{attribute 'linkalways'} 
{attribute 'no_explicit_call' := 'This FB is a CLASS and must be accessed using methods or properties'}
{attribute 'enable_dynamic_creation'}
FUNCTION_BLOCK Node_F_VN_VarianceFilterExp EXTENDS VisionNode
VAR
    ipSrcImage : _ITcVnImage;
    ipDestImage : _ITcVnImage;
    nKernelSize : _UDINT(0);
    fScale : _LREAL(1.0);
    eBorderType : _ETcVnBorderInterpolationMethod(ETcVnBorderInterpolationMethod.TCVN_BIM_DEFAULT);
    hrPrev : _HRESULT(S_OK);
	hresult : _HRESULT(S_OK);
END_VAR

METHOD PUBLIC  Clone : I_Node
VAR
	pNode : POINTER TO Node_F_VN_VarianceFilterExp;
END_VAR
pNode := __NEW(Node_F_VN_VarianceFilterExp);
Clone := pNode^;
END_METHOD

METHOD FB_init : BOOL
VAR_INPUT
	bInitRetains : BOOL; // if TRUE, the retain variables are initialized (warm start / cold start)
	bInCopyCode : BOOL;  // if TRUE, the instance afterwards gets moved into the copy code (online change)
END_VAR
AddInput('ipSrcImage', ipSrcImage);
AddParameter('nKernelSize', nKernelSize);
AddParameter('fScale', fScale);
AddParameter('eBorderType', eBorderType);
AddInput('hrPrev', hrPrev);
AddOutput('ipDestImage', ipDestImage);
AddOutput('hresult',hresult);
END_METHOD

METHOD PROTECTED OnExecute
hresult.Value := F_VN_VarianceFilterExp(
    ipSrcImage := ipSrcImage.Value,
	ipDestImage := ipDestImage.Value,
    nKernelSize := nKernelSize.Value,
    fScale := fScale.Value,
    eBorderType := eBorderType.Value,
	hrPrev:= hrPrev.Value);
END_METHOD

METHOD PUBLIC PreExecutionCheck
VAR_INPUT
	Check : I_PreExecutionChecks;
END_VAR
Check.IsTrue(ipSrcImage.IsValid, 'ipSrcImage must contain an image');
Check.IsTrue(ipSrcImage.HasChannelCount(1), 'ipSrcImage must have 1 channel');
Check.IsTrue(ipSrcImage.IsPixelDepth(8), 'ipSrcImage must have 8 bit pixel depth');
END_METHOD

END_FUNCTION_BLOCK

(* stored: Version 1.1.0.1, ProductVersion 3.1.4024.15
   POU Node_F_VN_VarianceFilterExp: Id {ec72eb1b-c208-0201-29da-b8ee69a8bbda}, SpecialFunc None
   Folder Constructor: Id {8adafb91-adce-084b-2e91-cef4613236de}
   Method Clone: Id {662ff759-926a-0ebd-327f-108780fea957}
   Method FB_init: Id {ce8accd2-94ad-0059-333f-8b95a5f727de}
   Method OnExecute: Id {6ef2bfa2-f868-09f1-2f95-a6ef78557b24}
   Method PreExecutionCheck: Id {ecd54f4f-1023-07f3-3d19-507725de6dd3} *)
